CASE eMode OF
//	====================================================================PRODUCTION MODE=========================================================	
	E_PMLUnitMode.ePMLUnitMode_Production:			
		;
//	====================================================================MANUAL MODE=============================================================	
	E_PMLUnitMode.ePMLUnitMode_Manual:				
		;
//	=====================================================================MAINTENANCE MODE=======================================================	
	E_PMLUnitMode.ePMLUnitMode_Maintenance:			
		;	
//	=====================================================================CUSTOM MODE 1==========================================================	
(*	E_PMLUnitMode.ePMLUnitMode_YOURCUSTOMMODE		
		;*)
//	======================================================================INVALID MODE==========================================================	
	E_PMLUnitMode.ePMLUnitMode_Invalid:				
		;
END_CASE
*)
END_METHOD

METHOD Suspending
//bNoStateTasksToComplete := TRUE;		// Change to False if not used

//Implement state Tasks here
(*
IF (insert your completion conditions) THEN

bStateTasksComplete := TRUE;				//Once these actions are completed successfully, set bStateTasksComplete to allow the base code to advance once all children have also reached the proper state

END_IF
*)

SUPER^.Suspending();

(*	Reference State Machine for mode specific actions - Be sure to paste above the SUPER^ Call if used - Delete if not needed

CASE eMode OF
//	====================================================================PRODUCTION MODE=========================================================	
	E_PMLUnitMode.ePMLUnitMode_Production:			
		;
//	====================================================================MANUAL MODE=============================================================	
	E_PMLUnitMode.ePMLUnitMode_Manual:				
		;
//	=====================================================================MAINTENANCE MODE=======================================================	
	E_PMLUnitMode.ePMLUnitMode_Maintenance:			
		;	
//	=====================================================================CUSTOM MODE 1==========================================================	
(*	E_PMLUnitMode.ePMLUnitMode_YOURCUSTOMMODE		
		;*)
//	======================================================================INVALID MODE==========================================================	
	E_PMLUnitMode.ePMLUnitMode_Invalid:				
		;
END_CASE
*)
END_METHOD

METHOD Unholding
//bNoStateTasksToComplete := TRUE;		// Change to False if not used

//Implement state Tasks here
(*
IF (insert your completion conditions) THEN

bStateTasksComplete := TRUE;				//Once these actions are completed successfully, set bStateTasksComplete to allow the base code to advance once all children have also reached the proper state

END_IF
*)

SUPER^.Unholding();

(*	Reference State Machine for mode specific actions - Be sure to paste above the SUPER^ Call if used - Delete if not needed

CASE eMode OF
//	====================================================================PRODUCTION MODE=========================================================	
	E_PMLUnitMode.ePMLUnitMode_Production:			
		;
//	====================================================================MANUAL MODE=============================================================	
	E_PMLUnitMode.ePMLUnitMode_Manual:				
		;
//	=====================================================================MAINTENANCE MODE=======================================================	
	E_PMLUnitMode.ePMLUnitMode_Maintenance:			
		;	
//	=====================================================================CUSTOM MODE 1==========================================================	
(*	E_PMLUnitMode.ePMLUnitMode_YOURCUSTOMMODE		
		;*)
//	======================================================================INVALID MODE==========================================================	
	E_PMLUnitMode.ePMLUnitMode_Invalid:				
		;
END_CASE
*)
END_METHOD

METHOD Unsuspending
//bNoStateTasksToComplete := TRUE;		// Change to False if not used

//Implement state Tasks here
(*
IF (insert your completion conditions) THEN

bStateTasksComplete := TRUE;				//Once these actions are completed successfully, set bStateTasksComplete to allow the base code to advance once all children have also reached the proper state

END_IF
*)

SUPER^.Unsuspending();

(*	Reference State Machine for mode specific actions - Be sure to paste above the SUPER^ Call if used - Delete if not needed

CASE eMode OF
//	====================================================================PRODUCTION MODE=========================================================	
	E_PMLUnitMode.ePMLUnitMode_Production:			
		;
//	====================================================================MANUAL MODE=============================================================	
	E_PMLUnitMode.ePMLUnitMode_Manual:				
		;
//	=====================================================================MAINTENANCE MODE=======================================================	
	E_PMLUnitMode.ePMLUnitMode_Maintenance:			
		;	
//	=====================================================================CUSTOM MODE 1==========================================================	
(*	E_PMLUnitMode.ePMLUnitMode_YOURCUSTOMMODE		
		;*)
//	======================================================================INVALID MODE==========================================================	
	E_PMLUnitMode.ePMLUnitMode_Invalid:				
		;
END_CASE
*)
END_METHOD

METHOD Aborted
CASE eMode OF
//	====================================================================PRODUCTION MODE=========================================================	
	E_PMLUnitMode.ePMLUnitMode_Production:			
		;
//	====================================================================MANUAL MODE=============================================================	
	E_PMLUnitMode.ePMLUnitMode_Manual:				
		;
//	=====================================================================MAINTENANCE MODE=======================================================	
	E_PMLUnitMode.ePMLUnitMode_Maintenance:			
		;	
//	=====================================================================CUSTOM MODE 1==========================================================	
(*	E_PMLUnitMode.ePMLUnitMode_YOURCUSTOMMODE		
		;*)
//	======================================================================INVALID MODE==========================================================	
	E_PMLUnitMode.ePMLUnitMode_Invalid:				
		;
END_CASE
END_METHOD

METHOD Complete
CASE eMode OF
//	====================================================================PRODUCTION MODE=========================================================	
	E_PMLUnitMode.ePMLUnitMode_Production:			
		;
//	====================================================================MANUAL MODE=============================================================	
	E_PMLUnitMode.ePMLUnitMode_Manual:				
		;
//	=====================================================================MAINTENANCE MODE=======================================================	
	E_PMLUnitMode.ePMLUnitMode_Maintenance:			
		;	
//	=====================================================================CUSTOM MODE 1==========================================================	
(*	E_PMLUnitMode.ePMLUnitMode_YOURCUSTOMMODE		
		;*)
//	======================================================================INVALID MODE==========================================================	
	E_PMLUnitMode.ePMLUnitMode_Invalid:				
		;
END_CASE
END_METHOD

METHOD Execute
CASE eMode OF
//	====================================================================PRODUCTION MODE=========================================================	
	E_PMLUnitMode.ePMLUnitMode_Production:			
		;
//	====================================================================MANUAL MODE=============================================================	
	E_PMLUnitMode.ePMLUnitMode_Manual:				
		;
//	=====================================================================MAINTENANCE MODE=======================================================	
	E_PMLUnitMode.ePMLUnitMode_Maintenance:			
		;	
//	=====================================================================CUSTOM MODE 1==========================================================	
(*	E_PMLUnitMode.ePMLUnitMode_YOURCUSTOMMODE		
		;*)
//	======================================================================INVALID MODE==========================================================	
	E_PMLUnitMode.ePMLUnitMode_Invalid:				
		;
END_CASE
END_METHOD

METHOD Held
CASE eMode OF
//	====================================================================PRODUCTION MODE=========================================================	
	E_PMLUnitMode.ePMLUnitMode_Production:			
		;
//	====================================================================MANUAL MODE=============================================================	
	E_PMLUnitMode.ePMLUnitMode_Manual:				
		;
//	=====================================================================MAINTENANCE MODE=======================================================	
	E_PMLUnitMode.ePMLUnitMode_Maintenance:			
		;	
//	=====================================================================CUSTOM MODE 1==========================================================	
(*	E_PMLUnitMode.ePMLUnitMode_YOURCUSTOMMODE		
		;*)
//	======================================================================INVALID MODE==========================================================	
	E_PMLUnitMode.ePMLUnitMode_Invalid:				
		;
END_CASE
END_METHOD

METHOD Idle
CASE eMode OF
//	====================================================================PRODUCTION MODE=========================================================	
	E_PMLUnitMode.ePMLUnitMode_Production:			
		;
//	====================================================================MANUAL MODE=============================================================	
	E_PMLUnitMode.ePMLUnitMode_Manual:				
		;
//	=====================================================================MAINTENANCE MODE=======================================================	
	E_PMLUnitMode.ePMLUnitMode_Maintenance:			
		;	
//	=====================================================================CUSTOM MODE 1==========================================================	
(*	E_PMLUnitMode.ePMLUnitMode_YOURCUSTOMMODE		
		;*)
//	======================================================================INVALID MODE==========================================================	
	E_PMLUnitMode.ePMLUnitMode_Invalid:				
		;
END_CASE
END_METHOD

METHOD Stopped
CASE eMode OF
//	====================================================================PRODUCTION MODE=========================================================	
	E_PMLUnitMode.ePMLUnitMode_Production:			
		;
//	====================================================================MANUAL MODE=============================================================	
	E_PMLUnitMode.ePMLUnitMode_Manual:				
		;
//	=====================================================================MAINTENANCE MODE=======================================================	
	E_PMLUnitMode.ePMLUnitMode_Maintenance:			
		;	
//	=====================================================================CUSTOM MODE 1==========================================================	
(*	E_PMLUnitMode.ePMLUnitMode_YOURCUSTOMMODE		
		;*)
//	======================================================================INVALID MODE==========================================================	
	E_PMLUnitMode.ePMLUnitMode_Invalid:				
		;
END_CASE
END_METHOD

METHOD Suspended
CASE eMode OF
//	====================================================================PRODUCTION MODE=========================================================	
	E_PMLUnitMode.ePMLUnitMode_Production:			
		;
//	====================================================================MANUAL MODE=============================================================	
	E_PMLUnitMode.ePMLUnitMode_Manual:				
		;
//	=====================================================================MAINTENANCE MODE=======================================================	
	E_PMLUnitMode.ePMLUnitMode_Maintenance:			
		;	
//	=====================================================================CUSTOM MODE 1==========================================================	
(*	E_PMLUnitMode.ePMLUnitMode_YOURCUSTOMMODE		
		;*)
//	======================================================================INVALID MODE==========================================================	
	E_PMLUnitMode.ePMLUnitMode_Invalid:				
		;
END_CASE
END_METHOD

METHOD Undefined
CASE eMode OF
//	====================================================================PRODUCTION MODE=========================================================	
	E_PMLUnitMode.ePMLUnitMode_Production:			
		;
//	====================================================================MANUAL MODE=============================================================	
	E_PMLUnitMode.ePMLUnitMode_Manual:				
		;
//	=====================================================================MAINTENANCE MODE=======================================================	
	E_PMLUnitMode.ePMLUnitMode_Maintenance:			
		;	
//	=====================================================================CUSTOM MODE 1==========================================================	
(*	E_PMLUnitMode.ePMLUnitMode_YOURCUSTOMMODE		
		;*)
//	======================================================================INVALID MODE==========================================================	
	E_PMLUnitMode.ePMLUnitMode_Invalid:				
		;
END_CASE
END_METHOD

END_FUNCTION_BLOCK

// Base/02_Component/FB_ComponentBase
FUNCTION_BLOCK FB_ComponentBase IMPLEMENTS ITF_ComponentBase
VAR_INPUT
END_VAR
VAR_OUTPUT
END_VAR
VAR CONSTANT
	//Constant declarations
	COMPONENT_BASE_ALARM_COUNT	: UDINT := 16;
END_VAR

VAR	
	//ITF_BasicComponent internal property variables
	bError 			: BOOL;			//Boolean to signal that an error has ocurred
	nErrorID 		: UDINT;		//Integer ID to identify the proper alarm to be posted from the parent module
	bEnabled		: BOOL;			//Enables or disables the component
	bSimulate		: BOOL;			//TRUE disables all hardware I/O and simulates input and output behavior
	sName			: STRING;		//String name of the component
	bActive			: BOOL;			//TRUE when the component is in its energized state, motion or detection
	bReady			: BOOL;			//TRUE when the component is ready for operation - (Should be set in extended component based on specific hardware and operation of the given component)
	eCurrentAlarmSeverity	: TcEventSeverity;
	a_eParentFaultResponseDefinitions		: ARRAY[0..4] OF E_AlarmResponse := [	E_AlarmResponse.NoResponse,
																					E_AlarmResponse.NoResponse,
																					E_AlarmResponse.NoResponse,
																					E_AlarmResponse.Abort_ImmediateError,
																					E_AlarmResponse.Abort_ImmediateError];
	
	//Alarming
	a_fbComponentBaseAlarms : ARRAY[1..COMPONENT_BASE_ALARM_COUNT] OF FB_TcAlarm;
	
	//HMI Monitoring and control structure
	stComponentBaseHMI : ST_ComponentBase_HMI;
	
	//Internal Variables
	bInitialized	: BOOL;
	bResetHappenedThisScan	: BOOL;		//Used for catching reset loops where errors are set and cleared in the same scan, causing a spike in Disk and ADS usage
	bResetHappenedLastScan	: BOOL;
	sTemp					: STRING;	//Generic Temp string for messaging or wherever else it is needed	
END_VAR

PROPERTY Name : STRING
GET
Name := sName;
END_GET
SET
sName := Name;
END_SET
END_PROPERTY

PROPERTY ParentResponseDefinitions : ARRAY[0..4] OF E_AlarmResponse
GET
ParentResponseDefinitions[TcEventSeverity.Verbose] := a_eParentFaultResponseDefinitions[TcEventSeverity.Verbose];
ParentResponseDefinitions[TcEventSeverity.Info] := a_eParentFaultResponseDefinitions[TcEventSeverity.Info];
ParentResponseDefinitions[TcEventSeverity.Warning] := a_eParentFaultResponseDefinitions[TcEventSeverity.Warning];
ParentResponseDefinitions[TcEventSeverity.Error] := a_eParentFaultResponseDefinitions[TcEventSeverity.Error];
ParentResponseDefinitions[TcEventSeverity.Critical] := a_eParentFaultResponseDefinitions[TcEventSeverity.Critical];
END_GET
SET
a_eParentFaultResponseDefinitions[TcEventSeverity.Verbose] := ParentResponseDefinitions[TcEventSeverity.Verbose];
a_eParentFaultResponseDefinitions[TcEventSeverity.Info] := ParentResponseDefinitions[TcEventSeverity.Info];
a_eParentFaultResponseDefinitions[TcEventSeverity.Warning] := ParentResponseDefinitions[TcEventSeverity.Warning];
a_eParentFaultResponseDefinitions[TcEventSeverity.Error] := ParentResponseDefinitions[TcEventSeverity.Error];
a_eParentFaultResponseDefinitions[TcEventSeverity.Critical] := ParentResponseDefinitions[TcEventSeverity.Critical];
END_SET
END_PROPERTY


PROPERTY Simulate : BOOL
GET
Simulate := bSimulate;
END_GET
SET
bSimulate := Simulate;
END_SET
END_PROPERTY

PROPERTY Enabled : BOOL	//Enables or disables the component
GET
Enabled := bEnabled;
END_GET
SET
bEnabled := Enabled;
END_SET
END_PROPERTY

PROPERTY Active : BOOL	//TRUE when the component is in motion or otherwise completing a commanded task
GET
Active := bActive;
END_GET
END_PROPERTY

PROPERTY CurrentAlarmSeverity : TcEventSeverity
GET
CurrentAlarmSeverity := eCurrentAlarmSeverity;
END_GET
END_PROPERTY

PROPERTY Error : BOOL	//Boolean to signal that an error has ocurred
GET
Error := bError;
END_GET
END_PROPERTY

PROPERTY ErrorID : UDINT	//Integer ID to identify the proper alarm to be posted from the parent module
GET
ErrorID := nErrorID;
END_GET
SET
nErrorID := ErrorID;
END_SET
END_PROPERTY

PROPERTY Ready : BOOL
GET
Ready := bReady;
END_GET
END_PROPERTY

METHOD AllowHMIControl : BOOL
VAR_INPUT
END_VAR
stComponentBaseHMI.bHMIControlAvailable := TRUE;
END_METHOD

METHOD BlockHMIControl : BOOL
VAR_INPUT
END_VAR
stComponentBaseHMI.bHMIControlAvailable := FALSE;
END_METHOD

{attribute 'call_after_online_change_slot' := '<slot>'}
METHOD CreateEvents : BOOL
VAR_INPUT
END_VAR
F_CreateAllEventsInClass(	p_aAlarms := a_fbComponentBaseAlarms,
							nClassSize := SIZEOF(TC_EVENTS.ComponentBase),
							pInitEvent := ADR(TC_EVENTS.PMLAlarms.InitReferenceEvent),
							sPrefix := sName);
END_METHOD

METHOD CyclicLogic : BOOL		//Should be called Externally akin to the PML Modules
IF NOT bInitialized THEN
	initialize();
	bInitialized := TRUE;
END_IF

IF NOT bSimulate AND NOT bError THEN	//If not in simulation mode or error state
	StandardOperation();
ELSIF NOT bError THEN
	SimulateOperation();	//Simulate inputs and outputs
ELSE
	ErrorOperation();
END_IF

Monitoring();		//Constant error and status monitoring
HardwareUpdate();	//Passes internal commands to hardware outputs and vice versa for inputs, implement via extended FB override
HMICommunication();	//Keeps the HMI data up to date, and processes requests from the HMI for this component
END_METHOD

METHOD Reset : BOOL
IF bError (*AND NOT nErrorID = E_ComponentBase.ResetLoopDetected *)THEN
	bError := FALSE;
	nErrorID := 0;
	
	bResetHappenedThisScan := TRUE;
//ELSIF bError AND NOT a_fbComponentBaseAlarms[E_ComponentBase.ResetNotPermitted].bRaised THEN
//	a_fbComponentBaseAlarms[E_ComponentBase.ResetNotPermitted].Raise(0);
ELSIF NOT bError THEN
	;
END_IF
END_METHOD

METHOD ErrorOperation : BOOL
VAR_INPUT
END_VAR
//Override from extended FB with error operation logic (Shut off outputs, clear inputs, blink, send error messages, etc)
END_METHOD

METHOD HardwareUpdate : BOOL
VAR_INPUT
END_VAR
//override from extended FB with reads and writes between internal variables and hardware inputs and outputs
END_METHOD

METHOD HMICommunication : BOOL
//Extend this method in extended FBs to communicate specific implementation data

//Process HMI requests
IF stComponentBaseHMI.bIncomingHMIRequest AND NOT stComponentBaseHMI.bHMICommandConfirmation THEN		//If a request has been issued by the HMI, and a previous request has not just finished being processed
	IF stComponentBaseHMI.bHMIControlAvailable THEN		//If the current conditions permit HMI control (Should be determined by the extended application components)
		IF stComponentBaseHMI.bEnableHMIRequest THEN
			bEnabled := TRUE;
			stComponentBaseHMI.bHMICommandConfirmation := TRUE;	//Confirm that the request has been processed
		END_IF
		IF stComponentBaseHMI.bDisableHMIRequest THEN
			bEnabled := FALSE;
			stComponentBaseHMI.bHMICommandConfirmation := TRUE;	//Confirm that the request has been processed
		END_IF
		IF stComponentBaseHMI.bResetHMIRequest THEN
			Reset();
			stComponentBaseHMI.bHMICommandConfirmation := TRUE;	//Confirm that the request has been processed
		END_IF
		IF stComponentBaseHMI.bSimulateOperationHMIRequest THEN
			bSimulate := TRUE;
			stComponentBaseHMI.bHMICommandConfirmation := TRUE;	//Confirm that the request has been processed
		END_IF
		IF stComponentBaseHMI.bStandardOperationHMIRequest THEN
			bSimulate := FALSE;
			stComponentBaseHMI.bHMICommandConfirmation := TRUE;	//Confirm that the request has been processed
		END_IF
	END_IF
END_IF

//Update HMI status info
stComponentBaseHMI.bActive := bActive;
stComponentBaseHMI.bEnabled := bEnabled;
stComponentBaseHMI.sName := sName;
stComponentBaseHMI.bError := bError;
stComponentBaseHMI.bSimulate := bSimulate;
stComponentBaseHMI.nErrorID := nErrorID;
END_METHOD

METHOD initialize : BOOL
VAR_INPUT
END_VAR

VAR
	sTemp: STRING;
END_VAR
//Extend initialize as needed in extended FBs

sTemp := CONCAT(CONCAT(CONCAT('Component ', ': '), sName), ' '); 	//Creates a utility string for alarms and other messaging that reads (example text) - "Module 10 - Main Casepacker" to be followed by the alarm or message info
//TODO: Rename Event Class to AxisBase
F_CreateAllEventsInClass(	p_aAlarms := a_fbComponentBaseAlarms,
							nClassSize := SIZEOF(TC_EVENTS.ComponentBase),
							pInitEvent := ADR(TC_EVENTS.ComponentBase.InitReferenceEvent),
							sPrefix := sTemp );
END_METHOD

METHOD Monitoring : BOOL
VAR_INPUT
END_VAR
//Extend from extended FB with monitoring logic

//Used for catching reset loops where errors are set and cleared in the same scan, causing a spike in Disk and ADS usage
//To implement, condition error setting with a check for bResetHappenedThisScan, raise the ResetLoopDetected event, and stop error detection for the component
IF bResetHappenedThisScan AND NOT bResetHappenedLastScan THEN
	bResetHappenedLastScan := TRUE;
	bResetHappenedThisScan :=FALSE;
ELSE
	IF bError THEN
		RaiseAlarmWithStrings(a_fbComponentBaseAlarms[E_ComponentBase.ResetLoopDetected], UDINT_TO_STRING(nErrorID), '');
	END_IF
	bResetHappenedLastScan := FALSE;
END_IF

IF NOT a_fbComponentBaseAlarms[E_ComponentBase.SimulationWarning].bRaised AND bSimulate THEN
	a_fbComponentBaseAlarms[E_ComponentBase.SimulationWarning].Raise(0);
ELSIF a_fbComponentBaseAlarms[E_ComponentBase.SimulationWarning].bRaised AND NOT bSimulate THEN
	a_fbComponentBaseAlarms[E_ComponentBase.SimulationWarning].Clear(0,0);
END_IF

eCurrentAlarmSeverity := TcEventSeverity.Verbose;

eCurrentAlarmSeverity := F_GetMaxSeverityRaised(	a_fbAlarms := a_fbComponentBaseAlarms,
													eCurrentSeverity := eCurrentAlarmSeverity);
END_METHOD

METHOD RaiseAlarm : BOOL
VAR_IN_OUT
	fbAlarm		: FB_TcAlarm;
END_VAR
F_RaiseAlarmAndSetFlags(fbAlarm := fbAlarm,
						bErrorFlag := bError,
						nErrorID := nErrorID);
END_METHOD

METHOD RaiseAlarmWithStrings : BOOL
VAR_IN_OUT
	fbAlarm		: FB_TcAlarm;	//Alarm to be raised
END_VAR
VAR_INPUT
	sString_1	: STRING;		//First String Parameter (The Name of this component will be applied first automatically)
	sString_2	: STRING;		//Second String Parameter
END_VAR
F_RaiseAlarmWithStringsAndFlags( 	fbAlarm := fbAlarm,
									bErrorFlag := bError,
									nErrorID := nErrorID,
									sString_1 := sName,
									sString_2 := sString_1,
									sString_3 := sString_2);
END_METHOD

METHOD SimulateOperation : BOOL
VAR_INPUT
END_VAR
//Override from extended FB with simulated operation logic
END_METHOD

METHOD StandardOperation : BOOL
VAR_INPUT
END_VAR
//Override from extended FB with normal operation logic
END_METHOD

END_FUNCTION_BLOCK

// Base/03_Utilities/01_Events/F_RaiseAlarmAndSetFlags
FUNCTION F_RaiseAlarmAndSetFlags : BOOL
VAR_IN_OUT
	fbAlarm			: FB_TcAlarm;	//Alarm to be raised
	bErrorFlag		: BOOL;			//Error flag to set (VAR_IN_OUT, put the variable you want the function to SET here)
	nErrorID		: UDINT;			//Error ID to set (VAR_IN_OUT, put the variable you want the function to SET here) - Will be set using the ID of the given fbAlarm
END_VAR

bErrorFlag	:= TRUE;
nErrorID := fbAlarm.nEventId;

fbAlarm.Raise(0);

END_FUNCTION

// Base/03_Utilities/01_Events/F_RaiseAlarmWithStringsAndFlags
FUNCTION F_RaiseAlarmWithStringsAndFlags : BOOL
VAR_IN_OUT
	fbAlarm			: FB_TcAlarm;	//Alarm to be raised
	bErrorFlag		: BOOL;			//Error flag to set (VAR_IN_OUT, put the variable you want the function to SET here)
	nErrorID		: UDINT;			//Error ID to set (VAR_IN_OUT, put the variable you want the function to SET here) - Will be set using the ID of the given fbAlarm
END_VAR
VAR_INPUT
	sString_1	: STRING;
	sString_2	: STRING;
	sString_3	: STRING;
END_VAR

fbAlarm.ipArguments.Clear();

bErrorFlag	:= TRUE;
nErrorID := fbAlarm.nEventId;

F_RaiseAlarmWithStringParameters(	fbAlarm :=  fbAlarm,
										sString_1 := sString_1, 
										sString_2 := sString_2,
										sString_3 := sString_3);

END_FUNCTION

// Base/03_Utilities/02_DataStructures/01_Tree/01_Tree_IndexBased/FB_Tree_IndexBased
FUNCTION_BLOCK FB_Tree_IndexBased IMPLEMENTS ITF_Tree_IndexBased
VAR_IN_OUT
	a_stNodes : ARRAY[0..63] OF ST_Tree_IndexBased_Node;
END_VAR
VAR_INPUT
	sHead : STRING;
END_VAR
VAR
	bInitialized 	: BOOL;
	nNodeCount 		: DINT;
	nNewNodeIndex	: DINT;
	nHeadIndex		: DINT;
	
	//"Temp" variables for use in AddNodeAsChildByName
	nParentIndex 	: DINT;
	nChildCount		: DINT;
END_VAR

IF NOT bInitialized THEN
	initialize();
END_IF

METHOD AddNodeAsChildByName : BOOL
VAR_INPUT
	sNewName 	: STRING;
	sParentName	: STRING;
END_VAR
nParentIndex := GetIndexByName(sParentName);		//Find the index value of the designated parent node
nChildCount := a_stNodes[nParentIndex].nChildCount;
IF nParentIndex >= 0 THEN	//If GetIndex was successful
	IF (a_stNodes[nParentIndex].nChildCount < 64) THEN	//TODO: Proper Constant bound definition	//If the parent is not at max child count
		a_stNodes[nNewNodeIndex].sName := sNewName;		//assign new node name to next empty node in list
		a_stNodes[nNewNodeIndex].nParent := nParentIndex;	//assign the parent node to the new child node
		a_stNodes[nNewNodeIndex].nDepth := a_stNodes[nParentIndex].nDepth + 1;
		a_stNodes[nParentIndex].a_nChildren[nChildCount] := nNewNodeIndex;		//assign the new node location as the next child in the parent
		nNewNodeIndex := nNewNodeIndex + 1;		//Increment to next empty node
		a_stNodes[nParentIndex].nChildCount := nChildCount + 1;
	END_IF
END_IF
END_METHOD

METHOD GetIndexByName : DINT
VAR_INPUT
	sName : STRING;
END_VAR
VAR
	i : DINT;
END_VAR
FOR i := 0 TO nNodeCount DO
	IF a_stNodes[i].sName = sName THEN
		GetIndexByName := i;
		RETURN;
	END_IF
END_FOR

GetIndexByName := -1;
END_METHOD

METHOD PRIVATE initialize : BOOL
VAR_INPUT
END_VAR
//nNodeCount := UPPER_BOUND(a_stNodes,1) - LOWER_BOUND(a_stNodes,1) + 1;
nNodeCount := 64;
IF nNodeCount >= 0 THEN
	nHeadIndex := 0;//LOWER_BOUND(a_stNodes,1);
	a_stNodes[nHeadIndex].sName := sHead;
	a_stNodes[nHeadIndex].nDepth := 0;
	a_stNodes[nHeadIndex].nParent := -1;
	nNewNodeIndex := nHeadIndex + 1;
END_IF
END_METHOD

END_FUNCTION_BLOCK

// Base/03_Utilities/03_Math/01_LREAL/F_LREAL_RoundToPlace
FUNCTION F_LREAL_RoundToPlace : LREAL
VAR_INPUT
	fIn		: LREAL;
	nPlaces	: DINT;
END_VAR
VAR
END_VAR

F_LREAL_RoundToPlace := DINT_TO_LREAL(LREAL_TO_DINT(fIn * (nPlaces * 10)))/(nPlaces * 10);

END_FUNCTION

// Base/01_PML/01_Module/05_Visualizations/V_MachineModule
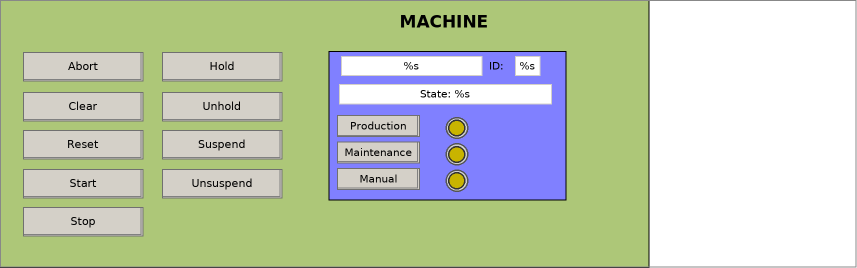
VISUALIZATION V_MachineModule  // 857x268
VAR_IN_OUT
	stVisu				: ST_PMLModuleBaseVISU;
END_VAR
    RoundedRectangle (0,0 649x268)
    Button (23,52 120x29), "Abort"
        tap stVisu.bAbortPressed
    Button (23,92 120x29), "Clear"
        tap stVisu.bClearPressed
    Button (23,130 120x29), "Reset"
        tap stVisu.bResetPressed
    Button (23,169 120x29), "Start"
        tap stVisu.bStartPressed
    Button (23,207 120x29), "Stop"
        tap stVisu.bStopPressed
    Button (162,52 120x29), "Hold"
        tap stVisu.bHoldPressed
    Button (162,92 120x29), "Unhold"
        tap stVisu.bUnholdPressed
    Button (162,130 120x29), "Suspend"
        tap stVisu.bSuspendPressed
    Button (162,169 120x29), "Unsuspend"
        tap stVisu.bUnsuspendPressed
    Frame (319,42 247x158)
        shows V_Module(stVisu := stVisu)
    Label (31,3 826x37), "MACHINE"
END_VISUALIZATION

// Base/01_PML/01_Module/05_Visualizations/V_Module
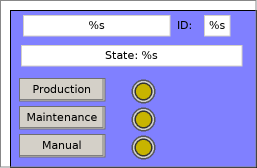
VISUALIZATION V_Module  // 257x168
VAR_IN_OUT
	stVisu				: ST_PMLModuleBaseVISU;
END_VAR
    RoundedRectangle (10,10 247x158)
    Textfield (23,15 147x21), "%s", text variable: stVisu.sModuleName
    Textfield (204,15 26x21), "%s", text variable: stVisu.nModuleID
    Label (165,14 39x23), "ID:"
    Textfield (21,45 221x21), "State: %s", text variable: stVisu.eState
    Button (19,78 86x23), "Production"
        tap stVisu.bProductionPressed
    Button (19,106 86x23), "Maintenance"
        tap stVisu.bMaintenancePressed
    Button (19,134 86x23), "Manual"
        tap stVisu.bManualPressed
    Lamp1 (130,78 27x27), variable: stVisu.eMode = E_PMLProtectedUnitMode.ePMLProtUnitMode_Production, style: Lamp-Lamp1-Yellow
    Lamp1 (130,106 27x27), variable: stVisu.eMode = E_PMLProtectedUnitMode.ePMLProtUnitMode_Maintenance, style: Lamp-Lamp1-Yellow
    Lamp1 (130,134 27x27), variable: stVisu.eMode = E_PMLProtectedUnitMode.ePMLProtUnitMode_Manual, style: Lamp-Lamp1-Yellow
END_VISUALIZATION
